{attribute addProperty BoxType "EL9520-0000-0016"}
{attribute addProperty Id "PowerOKAT %I*PowerOK_5B5BD03A810WcStateAT %I*WcState_98A4DF7520.250InfoDataAT %I*InfoData_192954DE1620"}
{attribute addProperty CRC "2241056452"}
{attribute addProperty SizeInBites "26"}
{attribute addProperty SizeInBytes "3.25"}
TYPE EL9520_B21A9EBB :
STRUCT
	{attribute addProperty Name "PowerOK"}
	PowerOK : PowerOK_5B5BD03A;
	{attribute addProperty Name "WcState"}
	WcState : WcState_98A4DF75;
	{attribute addProperty Name "InfoData"}
	InfoData : InfoData_192954DE;
END_STRUCT
END_TYPE

(* stored: Version 1.2.0.0, ProductVersion 3.1.4024.9
   DUT EL9520_B21A9EBB: Id {d0637558-7845-4668-9301-8a0be258a207} *)
